// TwinCAT 3 PLC project Untitled1
// ProgramVersion: 3.1.4024.0
// libraries:
//   Tc2_Standard, * (Beckhoff Automation GmbH)
//   Tc2_System, * (Beckhoff Automation GmbH)
//   Tc3_Module, * (Beckhoff Automation GmbH)
// project tree:
//   DUTs/ Location.TcDUT, Piece.TcDUT
//   GVLs/ GVL.TcGVL
//   / PlcTask.TcTTO
//   POUs/ AutomaticLogic_1.TcPOU, AutomationControl_1.TcPOU, Compressor.TcPOU, ManualControl.TcPOU, MotorControl.TcPOU, TrackingLogic.TcPOU, Vertical_process.TcPOU
// real-time tasks:
//   TASK PlcTask: cycle T#10ms, priority 20, ADS port 350
// I/O:
//   DEVICE Device 1 (EtherCAT), AmsNetId 5.132.85.181.2.1
//     Term 1 (EK1200) [EK1200-7000 EtherCAT Power supply (1,5A E-Bus)]
//       Term 2 (EL1859) [EL1859 8Ch. Dig. Input 24V, 3ms, 8Ch. Dig. Output 24V, 0.5A]
//       Term 3 (EL1859) [EL1859 8Ch. Dig. Input 24V, 3ms, 8Ch. Dig. Output 24V, 0.5A]
//       Term 4 (EL9011) [EL9011 End Terminal]
//   DEVICE Device 2 (NOV-DP-RAM)
//   DEVICE Device 3 (CX7000), AmsNetId 5.132.85.181.4.1
//     Term 1 (CX7028) [CX7028-0000-0118]
//       modules: Module 1 (DIO_2x), Module 3 (DIO_2x), Module 5 (DI_2x), Module 7 (DI_2x)
// variable links:
//   Untitled1/Untitled1 Instance <-> Device 1 (EtherCAT)/Term 1 (EK1200)/Term 2 (EL1859)
//     PlcTask Inputs/GVL.Limit1 <-> Channel 2/Input
//     PlcTask Inputs/GVL.Limit2 <-> Channel 5/Input
//     PlcTask Inputs/GVL.Sensor1 <-> Channel 1/Input
//     PlcTask Inputs/GVL.Sensor2 <-> Channel 6/Input
//     PlcTask Outputs/GVL.Compressor <-> Channel 9/Output
//     PlcTask Outputs/GVL.MotorRotate <-> Channel 14/Output
//     PlcTask Outputs/GVL.Piston1Back <-> Channel 11/Output
//     PlcTask Outputs/GVL.Piston2Back <-> Channel 16/Output
//     PlcTask Outputs/GVL.Piston1For <-> Channel 10/Output
//     PlcTask Outputs/GVL.Piston2For <-> Channel 15/Output
//     PlcTask Outputs/GVL.PistonVert <-> Channel 12/Output
//   Untitled1/Untitled1 Instance <-> Device 1 (EtherCAT)/Term 1 (EK1200)/Term 3 (EL1859)
//     PlcTask Outputs/GVL.MotorCon <-> Channel 10/Output
//   Untitled1/Untitled1 Instance <-> Device 3 (CX7000)/Term 1 (CX7028)
//     PlcTask Inputs/GVL.BlackBottomL <-> Module 5 (DI_2x)/DI_2x Input Channel 1/Input
//     PlcTask Inputs/GVL.BlackBottomR <-> Module 5 (DI_2x)/DI_2x Input Channel 2/Input
//     PlcTask Inputs/GVL.BlackTopL <-> Module 1 (DIO_2x)/DIO_2x Inputs Channel 2/Input
//     PlcTask Inputs/GVL.BlackTopR <-> Module 3 (DIO_2x)/DIO_2x Input Channel 1/Input
//     PlcTask Inputs/GVL.GrnBtn <-> Module 3 (DIO_2x)/DIO_2x Input Channel 2/Input
//     PlcTask Inputs/GVL.RedBtn <-> Module 1 (DIO_2x)/DIO_2x Inputs Channel 1/Input
//     PlcTask Inputs/GVL.Switch <-> Module 7 (DI_2x)/DI_2x Inputs Channel 1/Input
//     PlcTask Outputs/GVL.LEDGreen <-> Module 3 (DIO_2x)/DIO_2x Outputs Channel 1/Output
//     PlcTask Outputs/GVL.LEDRed <-> Module 1 (DIO_2x)/DIO_2x Outputs Channel 1/Output
//     PlcTask Outputs/GVL.LedBlueTop <-> Module 1 (DIO_2x)/DIO_2x Outputs Channel 2/Output

CONFIGURATION Untitled1
    RESOURCE PLC ON TwinCAT3
        TASK PlcTask(INTERVAL := T#10ms, PRIORITY := 20);
        PROGRAM AutomaticLogic_1 WITH PlcTask : AutomaticLogic_1;
    END_RESOURCE
END_CONFIGURATION

// ---- DUTs/Location.TcDUT
TYPE Location :
STRUCT
	Piece: Piece;
	Done: BOOL := FALSE;
	Occupied: BOOL := FALSE;
	Processed: BOOL := FALSE;
END_STRUCT
END_TYPE

// ---- DUTs/Piece.TcDUT
TYPE Piece :
STRUCT
	Id: INT := -1;
	Recipe: INT; // == Number of pushes
	Processed: INT := 0; 
END_STRUCT
END_TYPE

// ---- GVLs/GVL.TcGVL
{attribute 'qualified_only'}
VAR_GLOBAL
	Switch AT %I* : BOOL;
	LEDRed AT %Q* : BOOL;
	GrnBtn AT %I* : BOOL;
	LEDGreen AT %Q* : BOOL;
	RedBtn AT %I* : BOOL;
	LedBlueTop AT %Q* : BOOL;
	
	Compressor AT %Q* :BOOL; 
	Piston1For AT %Q* :BOOL := FALSE;
	Piston1Back AT %Q* :BOOL := FALSE;
	PistonVert AT %Q* :BOOL;
	MotorRotate AT %Q* :BOOL;
	Piston2For AT %Q* :BOOL;
	Piston2Back AT %Q* :BOOL;
	MotorCon AT %Q* :BOOL;
	
	BlackTopL AT %I* :BOOL;
	BlackTopR AT %I* :BOOL;
	BlackBottomL AT %I* :BOOL;
	BlackBottomR AT %I* :BOOL;
	
	Sensor1 AT %I* :BOOL;
	Limit1 AT %I* :BOOL;
	Limit2 AT %I* :BOOL;
	Sensor2 AT %I* :BOOL;
	
	Position : ARRAY [0..5] OF Location;
	
END_VAR

// ---- POUs/AutomaticLogic_1.TcPOU
PROGRAM AutomaticLogic_1
VAR
	Compressor1: Compressor;
	Tracking1: TrackingLogic;
	AutoCtrl: AutomationControl_1;
	Id_counter: CTU;
	Sensor1_FTrig: F_TRIG;
	lastP_trig: R_TRIG;
	limit1_trig: R_TRIG;
	
	activate: BOOL;
	vert_p: Vertical_process;
END_VAR

//AutoCtrl(piston1for := FALSE, piston1back := FALSE, piston2for := FALSE, piston2back := FALSE, pistonVert := FALSE, motorCon := FALSE, motorRotate := FALSE);
AutoCtrl();
Compressor1(switch:= GVL.Switch);
Tracking1();
Sensor1_FTrig(CLK:= GVL.Sensor1);
Id_counter();
lastP_trig(CLK := GVL.Sensor2);
Id_counter.CU := Sensor1_FTrig.Q;
limit1_trig(CLK:= GVL.Limit1);

vert_p(activate:= activate);


IF GVL.Switch = FALSE THEN
	
	//Init of Pieces
	IF Sensor1_FTrig.Q = TRUE THEN
		GVL.Position[0].Piece.Id := TO_INT(Id_counter.CV);
		GVL.Position[0].Piece.Recipe := 1;
		GVL.Position[0].Occupied := TRUE;
	END_IF
	
	// pushing from position 0
	IF (NOT GVL.Position[1].Occupied AND NOT AutoCtrl.motorRotate AND GVL.Position[0].Occupied) THEN
	AutoCtrl.piston1back := FALSE;	
	AutoCtrl.piston1for := TRUE;
		IF (GVL.Sensor1) THEN
			AutoCtrl.piston1for := FALSE;
			AutoCtrl.piston1back := TRUE;
			GVL.Position[0].Done := TRUE;
		END_IF
	END_IF

	// rotating table
	IF ((GVL.Position[1].Occupied AND NOT GVL.Position[2].Occupied AND NOT GVL.Position[3].Occupied) OR (NOT GVL.Position[1].Occupied AND (GVL.Position[2].Occupied AND GVL.Position[2].Processed) AND NOT GVL.Position[3].Occupied) OR (GVL.Position[1].Occupied AND (GVL.Position[2].Occupied AND GVL.Position[2].Processed) AND NOT GVL.Position[3].Occupied)) THEN
		AutoCtrl.motorRotate := TRUE;
		IF (GVL.Position[1].Occupied AND NOT GVL.Position[2].Occupied AND NOT GVL.Position[3].Occupied) THEN
			IF (GVL.Limit1) THEN
				AutoCtrl.motorRotate := FALSE;
				GVL.Position[1].Done := TRUE;
			END_IF	
		END_IF
		IF (NOT GVL.Position[1].Occupied AND (GVL.Position[2].Occupied AND GVL.Position[2].Processed)) THEN
			IF (GVL.Limit2) THEN
				AutoCtrl.motorRotate := FALSE;
				GVL.Position[2].Done := TRUE;
			END_IF
		END_IF
		IF (GVL.Position[1].Occupied AND (GVL.Position[2].Occupied AND GVL.Position[2].Processed) AND NOT GVL.Position[3].Occupied) THEN
			IF (GVL.Limit2) THEN
				AutoCtrl.motorRotate := FALSE;
				GVL.Position[2].Done := TRUE;
				IF (NOT GVL.Position[2].Done) THEN
					GVL.Position[1].Done := TRUE;
				END_IF
			END_IF
		END_IF
		
	END_IF
	
	// processing
	IF (GVL.Position[2].Occupied AND NOT GVL.Position[2].Processed) THEN
		IF (GVL.Position[2].Piece.Processed <= GVL.Position[2].Piece.Id + 1) THEN
			activate := TRUE;
			IF (vert_p.done) THEN
				//GVL.Position[2].Piece.Processed := GVL.Position[2].Piece.Processed + 1;
				activate := FALSE;
				IF (GVL.Position[2].Piece.Processed >= GVL.Position[2].Piece.Id +1) THEN
					GVL.Position[2].Processed := TRUE;
					//GVL.Position[2].Done := TRUE;
				END_IF
			END_IF
		END_IF
	END_IF
	
	// Piston 2
	IF (GVL.Position[3].Occupied AND NOT GVL.Position[4].Occupied) THEN
		
		AutoCtrl.piston2for := FALSE;
		AutoCtrl.piston2back := TRUE;	
		IF (NOT GVL.Limit2) THEN
			AutoCtrl.piston2back := FALSE;
			AutoCtrl.piston2for := TRUE;
			GVL.Position[3].Done := TRUE;
		END_IF
	END_IF
	
	// motorCon
	IF (GVL.Position[4].Occupied AND NOT GVL.Position[5].Occupied) THEN
		AutoCtrl.motorCon := TRUE;
		IF (NOT GVL.Sensor2) THEN
			AutoCtrl.motorCon := FALSE;
			GVL.Position[4].Done := TRUE;
		END_IF
	END_IF
	
	// LaSt position
	IF (lastP_trig.Q) THEN
		GVL.Position[5].Done := TRUE;
	END_IF

	
END_IF

END_PROGRAM

// ---- POUs/Compressor.TcPOU
FUNCTION_BLOCK Compressor
VAR_INPUT
	switch: BOOL;
	
END_VAR
VAR_OUTPUT
END_VAR
VAR
	R_TRIG_0: R_TRIG;
	R_TRIG0: BOOL;
	R_TRIG_1: R_TRIG;
	R_TRIG1: BOOL;
	R_TRIG_2: R_TRIG;
	R_TRIG2: BOOL;
END_VAR


R_TRIG_0(CLK := GVL.GrnBtn, Q=> R_TRIG0);
R_TRIG_1(CLK := GVL.REDBtn, Q=> R_TRIG1);
R_TRIG_2(CLK := GVL.Switch, Q=> R_TRIG2);

IF R_TRIG2 = TRUE THEN
	GVL.Compressor := FALSE;
END_IF


IF switch = FALSE THEN
	GVL.Compressor := TRUE;
ELSE

	IF  R_TRIG0 = TRUE THEN
		GVL.Compressor := TRUE;
	END_IF
	IF  R_TRIG1 = TRUE THEN
		GVL.Compressor := FALSE;
	END_IF 
	
END_IF;

END_FUNCTION_BLOCK

// ---- POUs/TrackingLogic.TcPOU
FUNCTION_BLOCK TrackingLogic
VAR_INPUT
END_VAR
VAR_OUTPUT
END_VAR
VAR
END_VAR



IF GVL.Position[0].Occupied  THEN
	IF GVL.Position[0].Done THEN
		GVL.Position[0].Done := FALSE;
		GVL.Position[1].Piece := GVL.Position[0].Piece;
		GVL.Position[1].Occupied := TRUE;
		GVL.Position[0].Occupied := FALSE;
		GVL.Position[1].Done := FALSE;
	END_IF
END_IF

IF GVL.Position[1].Occupied  THEN
	IF GVL.Position[1].Done THEN
		GVL.Position[1].Done := FALSE;
		GVL.Position[2].Piece := GVL.Position[1].Piece;
		GVL.Position[2].Occupied := TRUE;
		GVL.Position[1].Occupied := FALSE;
		GVL.Position[2].Done := FALSE;
		GVL.Position[2].Processed := FALSE;
	END_IF
END_IF

IF GVL.Position[2].Occupied  THEN
	IF GVL.Position[2].Done THEN
		//GVL.Position[2].Processed := FALSE;
		GVL.Position[3].Done := FALSE;
		GVL.Position[2].Occupied := FALSE;
		GVL.Position[3].Piece := GVL.Position[2].Piece;
		GVL.Position[3].Occupied := TRUE;
		GVL.Position[2].Done := FALSE;
	END_IF
END_IF

IF GVL.Position[3].Occupied  THEN
	IF GVL.Position[3].Done THEN
		GVL.Position[3].Done := FALSE;
		GVL.Position[4].Piece := GVL.Position[3].Piece;
		GVL.Position[4].Occupied := TRUE;
		GVL.Position[3].Occupied := FALSE;
		GVL.Position[4].Done := FALSE;
	END_IF
END_IF

IF GVL.Position[4].Occupied  THEN
	IF GVL.Position[4].Done THEN
		GVL.Position[4].Done := FALSE;
		GVL.Position[5].Piece := GVL.Position[4].Piece;
		GVL.Position[5].Occupied := TRUE;
		GVL.Position[4].Occupied := FALSE;
		GVL.Position[5].Done := FALSE;
	END_IF
END_IF

IF GVL.Position[5].Occupied  THEN
	IF GVL.Position[5].Done THEN
		GVL.Position[5].Done := FALSE;
		GVL.Position[5].Occupied := FALSE;
	END_IF
END_IF

END_FUNCTION_BLOCK

// ---- POUs/AutomationControl_1.TcPOU
FUNCTION_BLOCK AutomationControl_1
VAR_INPUT
	piston1for: BOOL;
	piston1back: BOOL;
	
	piston2for: BOOL;
	piston2back: BOOL;
	
	pistonVert: BOOL;
	
	motorRotate: BOOL;
	
	motorCon: BOOL;
	
END_VAR
VAR
	sleeping1: sleep;
	sleeping2: sleep;
END_VAR


//Piston1
GVL.Piston1For := piston1for;
GVL.Piston1Back := piston1back;

//Piston2
GVL.Piston2For := piston2for;
GVL.Piston2Back := piston2back;

GVL.PistonVert := pistonVert;

GVL.MotorCon := motorCon;

GVL.MotorRotate := motorRotate;

END_FUNCTION_BLOCK

// ---- POUs/Vertical_process.TcPOU
FUNCTION_BLOCK Vertical_process
VAR_INPUT
	activate: BOOL;
END_VAR
VAR_OUTPUT
	done: BOOL;
END_VAR
VAR
	TOF_1: TOF;
	R_TRIG_0: R_TRIG;
	F_TRIG_0: F_TRIG;
	TOF_0: TOF;
END_VAR
VAR // added by the converter: edge detectors and wires of the graphical bodies
    _w1 : BOOL;
END_VAR

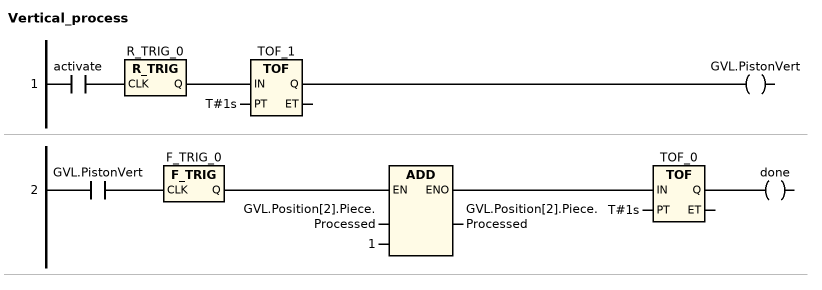
// NETWORK 1
R_TRIG_0(CLK := activate); // R_TRIG
TOF_1(IN := R_TRIG_0.Q, PT := T#1s); // TOF
GVL.PistonVert := TOF_1.Q;

// NETWORK 2
F_TRIG_0(CLK := GVL.PistonVert); // F_TRIG
_w1 := F_TRIG_0.Q;
IF _w1 THEN GVL.Position[2].Piece.Processed := GVL.Position[2].Piece.Processed + 1; END_IF
TOF_0(IN := _w1, PT := T#1s); // TOF
done := TOF_0.Q;

END_FUNCTION_BLOCK

// ---- POUs/ManualControl.TcPOU
PROGRAM ManualControl
VAR
	
	MotorControl: MotorControl;
	R_TRIG_0: R_TRIG;
	R_TRIG_1: R_TRIG;
	R_TRIG_2: R_TRIG;
	R_TRIG_3: R_TRIG;
	TON_0: TON;
	SR_0: SR;
	
	Compressor_0: Compressor;
END_VAR

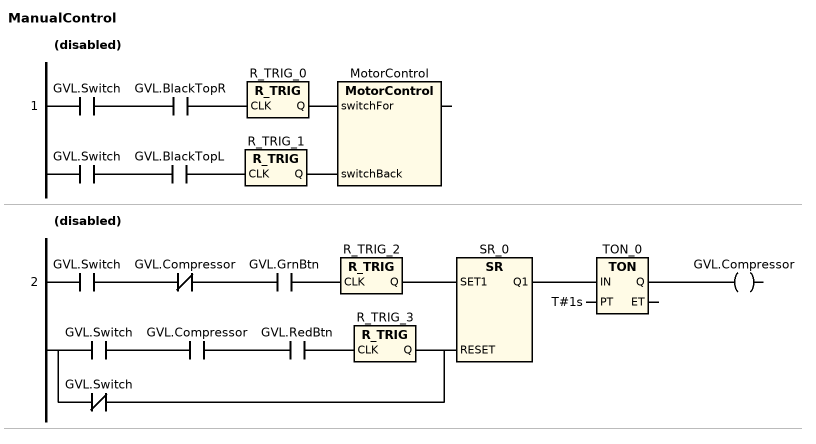
// NETWORK 1 (disabled)
// R_TRIG_0(CLK := GVL.Switch AND GVL.BlackTopR); // R_TRIG
// R_TRIG_1(CLK := GVL.Switch AND GVL.BlackTopL); // R_TRIG
// MotorControl(switchFor := R_TRIG_0.Q, switchBack := R_TRIG_1.Q);

// NETWORK 2 (disabled)
// R_TRIG_2(CLK := GVL.Switch AND NOT GVL.Compressor AND GVL.GrnBtn); // R_TRIG
// R_TRIG_3(CLK := GVL.Switch AND GVL.Compressor AND GVL.RedBtn); // R_TRIG
// SR_0(SET1 := R_TRIG_2.Q, RESET := R_TRIG_3.Q OR NOT GVL.Switch); // SR
// TON_0(IN := SR_0.Q1, PT := T#1s); // TON
// GVL.Compressor := TON_0.Q;

END_PROGRAM

// ---- POUs/MotorControl.TcPOU
FUNCTION_BLOCK MotorControl
VAR_INPUT
	switchFor: BOOL;
	switchBack: BOOL;
	
END_VAR
VAR_OUTPUT
END_VAR
VAR
	switchActive: BOOL;
	countValue: WORD;
	
	CounterMotor: CTUD;
	TOF_0: TOF;
	TOF_1: TOF;
	TOF_2: TOF;
	TOF_3: TOF;
	TOF_4: TOF;
	TOF_5: TOF;
	TOF_6: TOF;
	TON_0: TON;
END_VAR

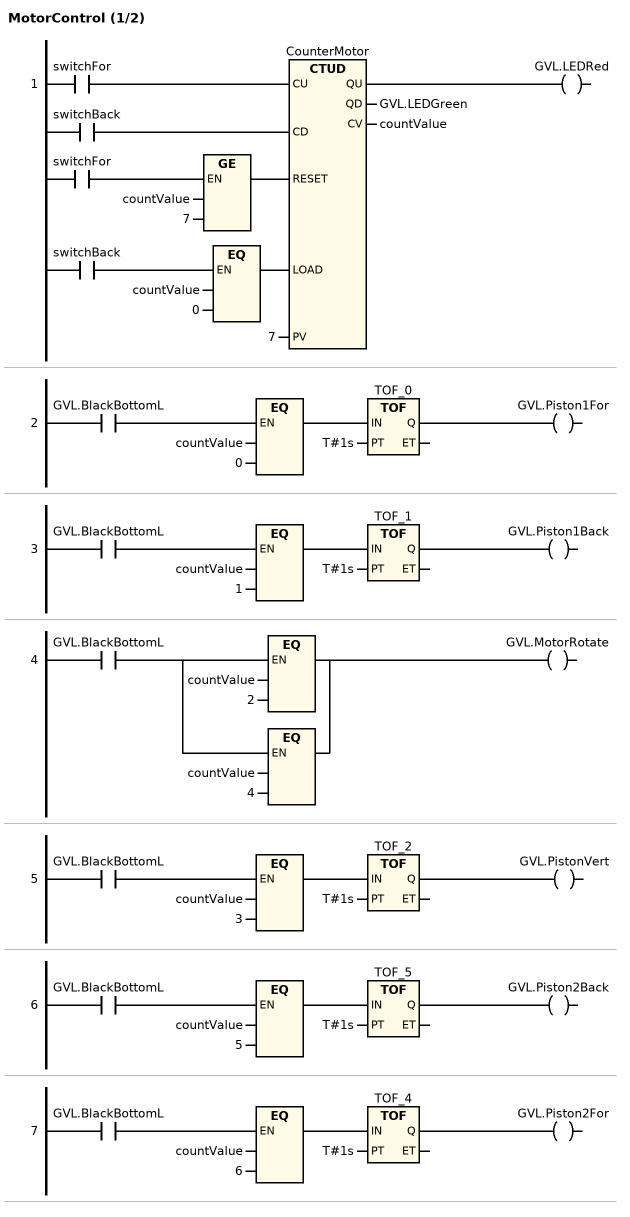
// NETWORK 1
CounterMotor(
    CU := switchFor,
    CD := switchBack,
    RESET := switchFor AND countValue >= 7,
    LOAD := switchBack AND countValue = 0,
    PV := 7,
    QD => GVL.LEDGreen,
    CV => countValue); // CTUD
GVL.LEDRed := CounterMotor.QU;

// NETWORK 2
TOF_0(IN := GVL.BlackBottomL AND countValue = 0, PT := T#1s); // TOF
GVL.Piston1For := TOF_0.Q;

// NETWORK 3
TOF_1(IN := GVL.BlackBottomL AND countValue = 1, PT := T#1s); // TOF
GVL.Piston1Back := TOF_1.Q;

// NETWORK 4
GVL.MotorRotate := GVL.BlackBottomL AND countValue = 2 OR GVL.BlackBottomL AND countValue = 4;

// NETWORK 5
TOF_2(IN := GVL.BlackBottomL AND countValue = 3, PT := T#1s); // TOF
GVL.PistonVert := TOF_2.Q;

// NETWORK 6
TOF_5(IN := GVL.BlackBottomL AND countValue = 5, PT := T#1s); // TOF
GVL.Piston2Back := TOF_5.Q;

// NETWORK 7
TOF_4(IN := GVL.BlackBottomL AND countValue = 6, PT := T#1s); // TOF
GVL.Piston2For := TOF_4.Q;

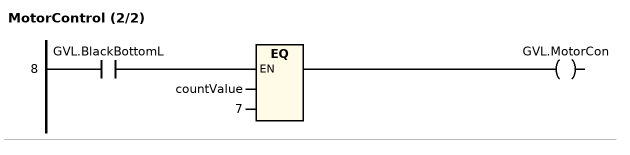
// NETWORK 8
GVL.MotorCon := GVL.BlackBottomL AND countValue = 7;

END_FUNCTION_BLOCK
